TYPE
  (* Standard: 61499-1 *)
  (* Version 1.0, 2026-07-21, Dimitrios Kalligaridis *)
  PACKAGE mypackage;
  Root : STRUCT
    middle : mypackage::Middle;
    id : BOOL;
  END_STRUCT;
END_TYPE
